// Mitsubishi GX Works2 project: Termin3_Treci_zadatak   PLC: FX3S

// task Task_01 (event TRUE, interval 0, priority 31): POU_01

PROGRAM POU_01
VAR
  S1_senzor : BOOL;
  broj_automobila : INT;
  S2_senzor : BOOL;
  izlaz_cmp : ARRAY [0..2] OF BOOL;
  crvena_lampa : BOOL;
  slobodnih_mesta : INT;
  izlaz_cmp_drugi : ARRAY [0..2] OF BOOL;
END_VAR
(* structured ladder/FBD written out as ST: instructions are called as NAME(EN, inputs, outputs); _pN, _eN, _tN stand for wires *)
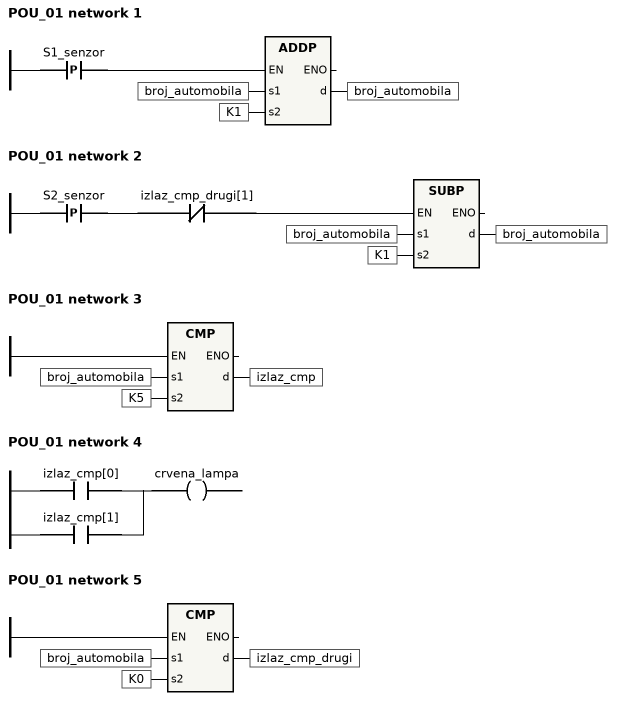
(* network 1 *)
ADDP(LDP(TRUE, S1_senzor), broj_automobila, K1, broj_automobila);
(* network 2 *)
SUBP(LDP(TRUE, S2_senzor) AND NOT izlaz_cmp_drugi[1], broj_automobila, K1, broj_automobila);
(* network 3 *)
CMP(TRUE, broj_automobila, K5, izlaz_cmp);
(* network 4 *)
crvena_lampa := izlaz_cmp[0] OR izlaz_cmp[1];
(* network 5 *)
CMP(TRUE, broj_automobila, K0, izlaz_cmp_drugi);
END_PROGRAM
